(* Schneider Machine Expert - Basic project memory floats, file version 2.0.0.0 *)
(* ProjectInformations: Name=New project *)

HARDWARE
  Cpu 0: TM221M16R/G
  EthernetConfiguration: NetworkName=M221, IpAllocationMode=FixedAddress, IpAddress=0.0.0.0, SubnetMask=0.0.0.0
  SerialLineConfiguration: Baud=Baud19200, Parity=ParityEven, DataBits=DataBits8, StopBits=StopBits1, PhysicalMedium=PhysicalMediumRs485, TransmissionMode=TransmissionModeModbusRtu, SlaveId=1, Addressing=SlaveAddressing
  MastTask: UsePeriodScanMode=false, PeriodScan=100
  FastTask: Period=255
  CpuBehavior: StartingMode=StartAsPreviousState, AutoSaveRamOnEeprom=true, WatchdogPeriod=250

SYMBOLS  (address, symbol, comment, settings)

POU New POU
  (* SectionNumber=1 *)

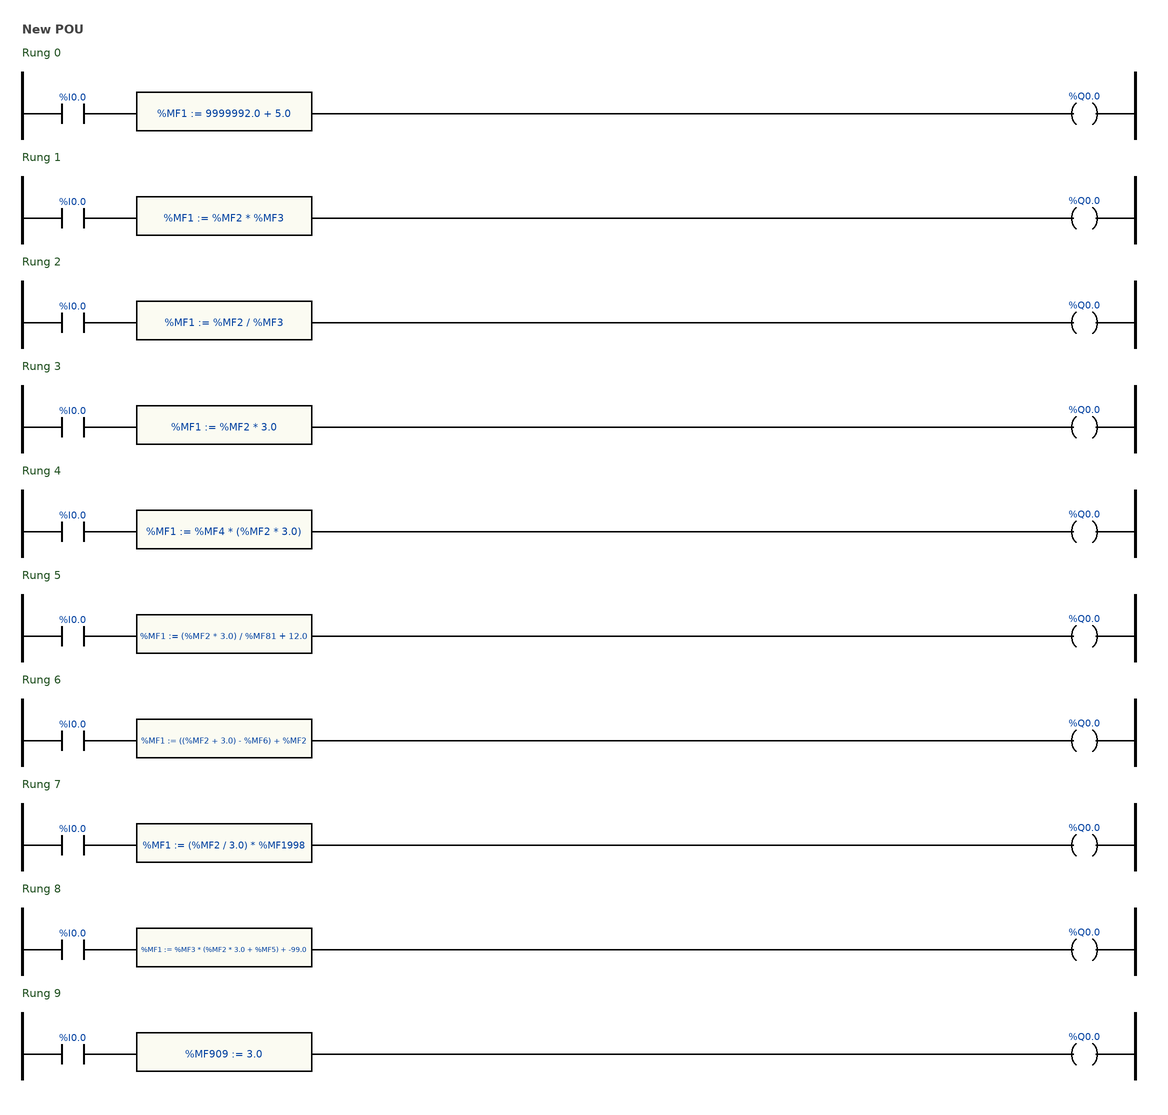

// Rung 0
  LD %I0.0
  OPER [ %MF1 := 9999992.0 + 5.0 ]
  ST %Q0.0
  // as ST:
  //   IF %I0.0 THEN %MF1 := 9999992.0 + 5.0; END_IF;
  //   %Q0.0 := %I0.0;

// Rung 1
  LD %I0.0
  OPER [ %MF1 := %MF2 * %MF3 ]
  ST %Q0.0
  // as ST:
  //   IF %I0.0 THEN %MF1 := %MF2 * %MF3; END_IF;
  //   %Q0.0 := %I0.0;

// Rung 2
  LD %I0.0
  OPER [ %MF1 := %MF2 / %MF3 ]
  ST %Q0.0
  // as ST:
  //   IF %I0.0 THEN %MF1 := %MF2 / %MF3; END_IF;
  //   %Q0.0 := %I0.0;

// Rung 3
  LD %I0.0
  OPER [ %MF1 := %MF2 * 3.0 ]
  ST %Q0.0
  // as ST:
  //   IF %I0.0 THEN %MF1 := %MF2 * 3.0; END_IF;
  //   %Q0.0 := %I0.0;

// Rung 4
  LD %I0.0
  OPER [ %MF1 := %MF4 * ( %MF2 * 3.0 ) ]
  ST %Q0.0
  // as ST:
  //   IF %I0.0 THEN %MF1 := %MF4 * ( %MF2 * 3.0 ); END_IF;
  //   %Q0.0 := %I0.0;

// Rung 5
  LD %I0.0
  OPER [ %MF1 := ( %MF2 * 3.0 ) / %MF81 + 12.0 ]
  ST %Q0.0
  // as ST:
  //   IF %I0.0 THEN %MF1 := ( %MF2 * 3.0 ) / %MF81 + 12.0; END_IF;
  //   %Q0.0 := %I0.0;

// Rung 6
  LD %I0.0
  OPER [ %MF1 := ( ( %MF2 + 3.0 ) - %MF6 ) + %MF2 ]
  ST %Q0.0
  // as ST:
  //   IF %I0.0 THEN %MF1 := ( ( %MF2 + 3.0 ) - %MF6 ) + %MF2; END_IF;
  //   %Q0.0 := %I0.0;

// Rung 7
  LD %I0.0
  OPER [ %MF1 := ( %MF2 / 3.0 ) * %MF1998 ]
  ST %Q0.0
  // as ST:
  //   IF %I0.0 THEN %MF1 := ( %MF2 / 3.0 ) * %MF1998; END_IF;
  //   %Q0.0 := %I0.0;

// Rung 8
  LD %I0.0
  OPER [ %MF1 := %MF3 * ( %MF2 * 3.0 + %MF5 ) + -99.0 ]
  ST %Q0.0
  // as ST:
  //   IF %I0.0 THEN %MF1 := %MF3 * ( %MF2 * 3.0 + %MF5 ) + -99.0; END_IF;
  //   %Q0.0 := %I0.0;

// Rung 9
  LD %I0.0
  OPER [ %MF909 := 3.0 ]
  ST %Q0.0
  // as ST:
  //   IF %I0.0 THEN %MF909 := 3.0; END_IF;
  //   %Q0.0 := %I0.0;

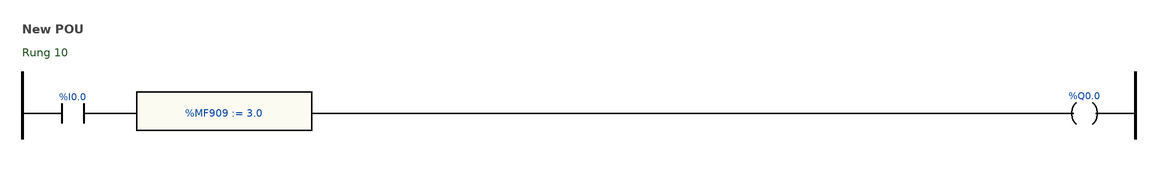

// Rung 10
  LD %I0.0
  OPER [ %MF909 := 3.0 ]
  ST %Q0.0
  // as ST:
  //   IF %I0.0 THEN %MF909 := 3.0; END_IF;
  //   %Q0.0 := %I0.0;
